Fanuc KAREL source: kf00116.KL

-- PROVISIONAL review KL for V1013-1; original PC SHA256 f494b5c816d7fa69f7f390490bc3570f9cd5b52fa6b626551d48377f6323faba
-- Incomplete behavior may be omitted. Consult companion uncertainty JSON. Do not deploy.
PROGRAM KF00116
%NOLOCKGROUP
BEGIN
  -- UNRESOLVED_PC offsets 0-1; opcodes 7B
  -- UNRESOLVED_PC offsets 6-19; opcodes 2D,9D,5A,79
  -- UNRESOLVED_PC offsets 24-29; opcodes 9D,7F
  -- UNRESOLVED_PC offsets 34-39; opcodes 7A
  -- UNRESOLVED_PC offsets 44-68; opcodes 2D,27,27,2D,9D,53,AA,54,7F
  -- UNRESOLVED_PC offsets 78-82; opcodes 7F
  -- UNRESOLVED_PC offsets 87-103; opcodes 27,27,2E,AA,23
  -- UNRESOLVED_PC offsets 108-112; opcodes 7F
END KF00116
